// TIA Portal V19 export
TYPE "VFD_Control"
   STRUCT
      NameplateSpeed : Real;
      AutoSpeedSP : Real;
      DriveIsRunning : Bool;
      ActualSpeed : Real;
      AxisActive : Bool;
      LockoutActive : Bool;
      ErrorPResent : Bool;
      HMI_VFD_Fault : Int;
      HMI_Error_Present : Bool;
      VFDFaultCode : Int;
      MotorState : Int;
      Actual_Current : Real;
      Actual_torque : Real;
      Peak_Current : Real;
      Peak_torque : Real;
   END_STRUCT;
END_TYPE
